TEXTLIST TextList_UpDownSlot_errorid
  0 = 'no_error'
  1 = 'not_connected'
  2 = 'invalid_state'
  3 = 'timeout_up'
  4 = 'timeout_down'
  5 = 'cmd_timeout'
  6 = 'io_error'
  7 = 'unknown_error'
  666 = 'emergency_error'
   = ''
END_TEXTLIST

(* stored: Version 1.1.0.1, ProductVersion 3.1.4024.11
   TextList TextList_UpDownSlot_errorid: Id {ff546c6a-49c1-4c3b-9118-92bf8ed8ecae} *)
